Omron Sysmac Studio project ToggleButton (Sysmac Studio 1.65.0.64007, StandardProject)

# Controller new_Controller_0: NX1P2-1040DT1 version 1.69
Task PrimaryTask (priority 4, period or condition 2000): Program0



PROGRAM Program0
VAR
    ToggleButton : BOOL;
    T1 : BOOL;
    T2 : BOOL;
    T3 : BOOL;
    T4 : BOOL;
    MotorCikis : BOOL;
END_VAR

(* Section Section0: ladder, written here as Structured Text *)

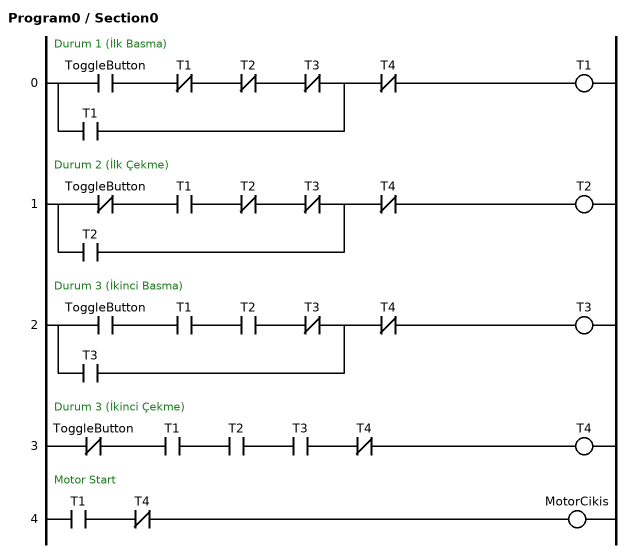
(* Rung 0: Durum 1 (İlk Basma) *)
T1 := ((ToggleButton AND NOT T1 AND NOT T2 AND NOT T3) OR T1) AND NOT T4;
(* Rung 1: Durum 2 (İlk Çekme) *)
T2 := ((NOT ToggleButton AND T1 AND NOT T2 AND NOT T3) OR T2) AND NOT T4;
(* Rung 2: Durum 3 (İkinci Basma) *)
T3 := ((ToggleButton AND T1 AND T2 AND NOT T3) OR T3) AND NOT T4;
(* Rung 3: Durum 3 (İkinci Çekme) *)
T4 := NOT ToggleButton AND T1 AND T2 AND T3 AND NOT T4;
(* Rung 4: Motor Start *)
MotorCikis := T1 AND NOT T4;
END_PROGRAM